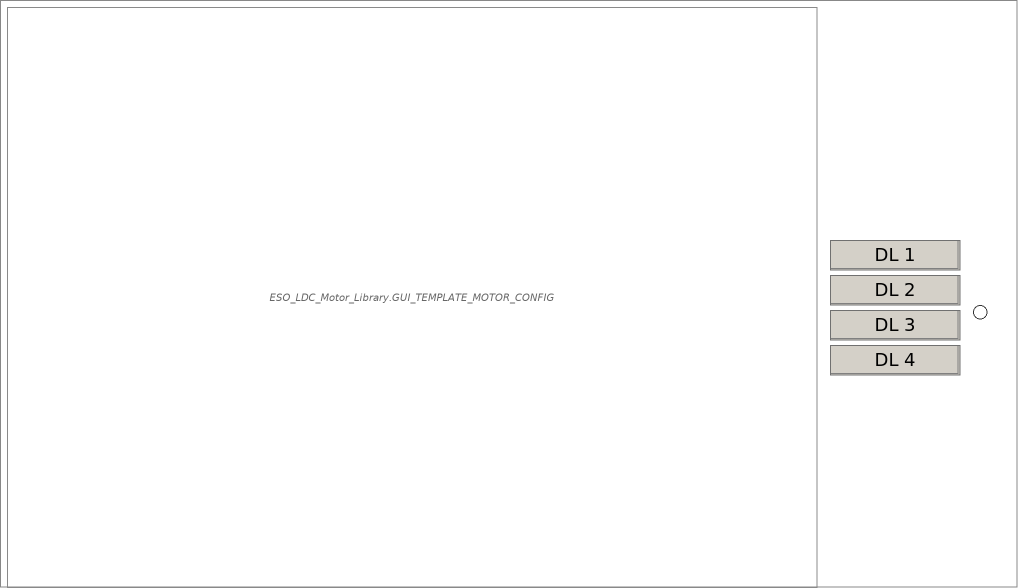
VISUALIZATION GUI_NOTT_DL_CONFIG  // 1018x588
    RadioButton (971,242 47x140), variable: MAIN.nott_ics.Delay_Lines.guiShutterIndex-1
        Areas[0]: Text=Radiobutton
        Areas[1]: Text=Radiobutton
    Button (830,240 130x30), "DL 1"
        OnMouseClick: execute { MAIN.nott_ics.Delay_Lines.guiShutterIndex := 1; }
    Button (830,275 130x30), "DL 2"
        OnMouseClick: execute { MAIN.nott_ics.Delay_Lines.guiShutterIndex := 2; }
    Button (830,310 130x30), "DL 3"
        OnMouseClick: execute { MAIN.nott_ics.Delay_Lines.guiShutterIndex := 3; }
    Button (830,345 130x30), "DL 4"
        OnMouseClick: execute { MAIN.nott_ics.Delay_Lines.guiShutterIndex := 4; }
    Frame (7,7 810x581)
        shows ESO_LDC_Motor_Library.GUI_TEMPLATE_MOTOR_CONFIG(m_Instance := MAIN.nott_ics.Delay_Lines.ptrDelayLines[MAIN.nott_ics.Delay_Lines.guiShutterIndex]^)
END_VISUALIZATION

(* stored: Version 1.1.0.1, ProductVersion 3.1.4024.12
   Visu GUI_NOTT_DL_CONFIG: Id {fbfe6e9d-3bd1-47ac-9852-3cb5a3405654} *)
